(* CoDeSys 2.3.9.48 project: LevelControlTanks.pro *)
(* Libraries: Standard.lib 8.11.10 11:37:48, SYSLIBCALLBACK.LIB 8.11.10 11:37:48 *)

(* PLC configuration (modules and I/O channels)
K-Bus [K_Bus] node 0, in %IB0 out %QB0
Fieldbus variables [FB_VARS] node 1, in %IB0 out %QB0
Flag variables [FLAG_VARS] node 2, in %IB0 out %QB0
Modbus-Master [MB_MASTER] node 3, in %IB0 out %QB0
*)

(* Global variable list: Global_Variables *)
VAR_GLOBAL
			(*VALVES*)
	InletValve: BOOL;
	ConnectingValve: BOOL;
	OutletValve: BOOL;
			(*SENSORS 1=high, 2=ok, 3=low*)
	Tank1Sensors: ARRAY[1..NumSensors] OF BOOL;
	Tank2Sensors: ARRAY[1..NumSensors] OF BOOL;
			(*FAULT*)
	faultSensors1: BOOL;
	faultSensors2: BOOL;

			(*SENSOR STATEMENT*)
	sensorStatementINTTank1: INT;
	sensorStatementINTTank2: INT;
	sensorString1: STRING;
	sensorString2: STRING;
END_VAR

VAR_GLOBAL CONSTANT
	NumSensors: INT := 3;
	NumTanks: INT := 2;
END_VAR

(* POU PLC_PRG, ST *)
PROGRAM PLC_PRG
VAR
END_VAR
TANK1;
TANK2;
TanksFault;
TanksInletValve;
TanksOutletValves;
END_PROGRAM

(* POU TANK1, ST *)
PROGRAM TANK1
VAR
	i: INT := 1;
	k: INT := 0;
END_VAR
	(*TANK1*)
FOR i := 1 TO 2 DO
	sensorStatementINTTank1 := sensorsStatement(HighSensor:= Tank1Sensors[1], OKSensor:=Tank1Sensors[2], LowSensor := Tank1Sensors[3]);
END_FOR;

(*
		INT VALUES TANKS
	1: TANK IS NOT FILLED
	2: TANK IS LOW WATER LEVEL
	3: SENSORS FAULT (LOW)
	4: TANK IS ON OK WATER LEVEL
	5: SENSORS FAULT (LOW AND OKAY)
	6: SENSORS FAULT (OKAY)
	7: TANK IS FULL ENOUGH
*)

		(*TANK1*)
IF sensorStatementINTTank1 = 1 THEN
	sensorString1:= 'Tank1 is empty';
END_IF;

IF sensorStatementINTTank1 = 2 THEN
	sensorString1:= 'Tank 1 is on low water level';
END_IF;

IF sensorStatementINTTank1 = 3 THEN
	sensorString1:= 'Sensor fault tank 1(LowSensor)';
END_IF;

IF sensorStatementINTTank1 = 4 THEN
	sensorString1:= 'Tank1 is on OK water level';
END_IF;

IF sensorStatementINTTank1 = 5 THEN
	sensorString1:= 'Sensor fault tank 1(LowSensor, OKsensor)';
END_IF;

IF sensorStatementINTTank1 = 6 THEN
	sensorString1:= 'Sensor fault tank 1(OKSensor)';
END_IF;

IF sensorStatementINTTank1 = 7 THEN
	sensorString1:= 'Tank1 is full enough';
END_IF;
END_PROGRAM

(* POU sensorsStatement, ST *)
FUNCTION sensorsStatement : INT
VAR_INPUT
	Highsensor: BOOL;
	OkSensor: BOOL;
	LowSensor: BOOL;
END_VAR
VAR
END_VAR
(*
		INT VALUES TANKS
	1: TANK IS NOT FILLED
	2: TANK IS LOW WATER LEVEL
	3: SENSORS FAULT (LOW)
	4: TANK IS ON OK WATER LEVEL
	5: SENSORS FAULT (LOW AND OKAY)
	6: SENSORS FAULT (OKAY)
	7: TANK IS FULL ENOUGH
*)

IF HighSensor = FALSE AND OkSensor = FALSE AND LowSensor = FALSE THEN
	sensorsStatement := 1;
END_IF;
IF HighSensor = FALSE AND OkSensor = FALSE AND LowSensor = TRUE THEN sensorsStatement := 2;END_IF;
IF HighSensor = FALSE AND OkSensor = TRUE AND LowSensor = FALSE THEN sensorsStatement := 3; END_IF;
IF HighSensor = FALSE AND OkSensor = TRUE AND LowSensor = TRUE THEN sensorsStatement := 4;  END_IF;
IF HighSensor = TRUE AND OkSensor = FALSE AND LowSensor = FALSE THEN sensorsStatement := 5;END_IF;
IF HighSensor = TRUE AND OkSensor = FALSE AND LowSensor = TRUE THEN sensorsStatement := 6;END_IF;
IF HighSensor = TRUE AND OkSensor = TRUE AND LowSensor = FALSE THEN sensorsStatement := 3; END_IF;
IF HighSensor = TRUE AND OkSensor = TRUE  AND LowSensor = TRUE  THEN sensorsStatement := 7; END_IF;
END_FUNCTION

(* POU TANK2, ST *)
PROGRAM TANK2
VAR
	j: INT := 1;
END_VAR
	(*TANK2*)
FOR j := 1 TO 2 DO
	sensorStatementINTTank2 := sensorsStatement(HighSensor:= Tank2Sensors[1], OKSensor:=Tank2Sensors[2], LowSensor := Tank2Sensors[3]);
END_FOR;

(*
		INT VALUES TANKS
	1: TANK IS NOT FILLED
	2: TANK IS LOW WATER LEVEL
	3: SENSORS FAULT (LOW)
	4: TANK IS ON OK WATER LEVEL
	5: SENSORS FAULT (LOW AND OKAY)
	6: SENSORS FAULT (OKAY)
	7: TANK IS FULL ENOUGH
*)

		(*TANK2*)
IF sensorStatementINTTank2 = 1 THEN
	sensorString2:= 'Tank2 is empty';
END_IF;

IF sensorStatementINTTank2  = 2 THEN
	sensorString2:= 'Tank 2 is on low water level';
END_IF;

IF sensorStatementINTTank2  = 3 THEN
	sensorString2:= 'Sensor fault tank 2(LowSensor)';
END_IF;

IF sensorStatementINTTank2  = 4 THEN
	sensorString2:= 'Tank2 is on OK water level';
END_IF;

IF sensorStatementINTTank2  = 5 THEN
	sensorString2:= 'Sensor fault tank 2(LowSensor, OKsensor)';
END_IF;

IF sensorStatementINTTank2  = 6 THEN
	sensorString2:= 'Sensor fault tank 2(OKSensor)';
END_IF;

IF sensorStatementINTTank2  = 7 THEN
	sensorString2:= 'Tank2 is full enough';
END_IF;
END_PROGRAM

(* POU FunctionBlocks/TanksFault, CFC *)
PROGRAM TanksFault
VAR
END_VAR
VAR (* helpers for the ST form of the networks *)
	_t30 : BOOL;
	_t8 : BOOL;
	_t41 : BOOL;
	_t39 : BOOL;
END_VAR
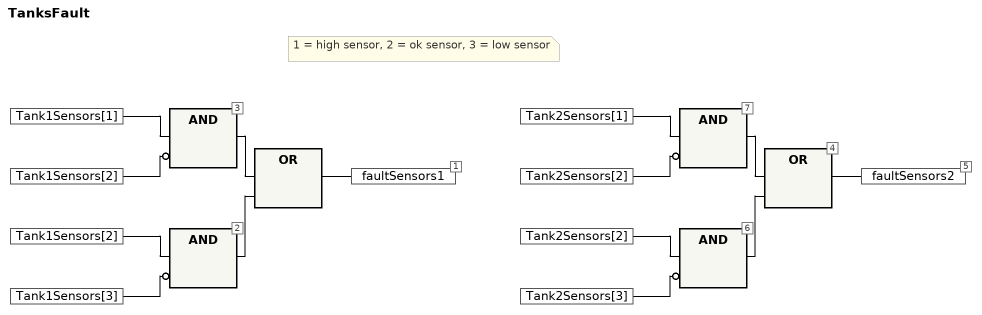
_CFC_ (* Continuous Function Chart, elements in execution order *)
(* 1 = high sensor, 2 = ok sensor, 3 = low sensor *)
#0 OR(#3, #2)
#1 faultSensors1 <= #0
#2 AND(Tank1Sensors[2], NOT Tank1Sensors[3])
#3 AND(Tank1Sensors[1], NOT Tank1Sensors[2])
#4 OR(#7, #6)
#5 faultSensors2 <= #4
#6 AND(Tank2Sensors[2], NOT Tank2Sensors[3])
#7 AND(Tank2Sensors[1], NOT Tank2Sensors[2])
_END_CFC_
(* the same logic as Structured Text *)
(* 1 = high sensor, 2 = ok sensor, 3 = low sensor *)
faultSensors1 := _t30 OR _t8;
_t8 := Tank1Sensors[2] AND NOT Tank1Sensors[3];
_t30 := Tank1Sensors[1] AND NOT Tank1Sensors[2];
faultSensors2 := _t41 OR _t39;
_t39 := Tank2Sensors[2] AND NOT Tank2Sensors[3];
_t41 := Tank2Sensors[1] AND NOT Tank2Sensors[2];
END_PROGRAM

(* POU FunctionBlocks/TanksInletValve, CFC *)
PROGRAM TanksInletValve
VAR
END_VAR
VAR (* helpers for the ST form of the networks *)
	_t30 : BOOL;
	_t8 : BOOL;
	_t52 : BOOL;
	_t50 : BOOL;
END_VAR
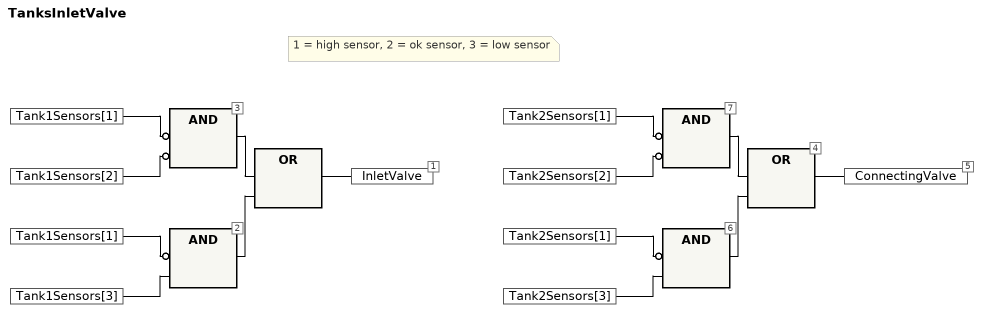
_CFC_ (* Continuous Function Chart, elements in execution order *)
(* 1 = high sensor, 2 = ok sensor, 3 = low sensor *)
#0 OR(#3, #2)
#1 InletValve <= #0
#2 AND(NOT Tank1Sensors[1], Tank1Sensors[3])
#3 AND(NOT Tank1Sensors[1], NOT Tank1Sensors[2])
#4 OR(#7, #6)
#5 ConnectingValve <= #4
#6 AND(NOT Tank2Sensors[1], Tank2Sensors[3])
#7 AND(NOT Tank2Sensors[1], NOT Tank2Sensors[2])
_END_CFC_
(* the same logic as Structured Text *)
(* 1 = high sensor, 2 = ok sensor, 3 = low sensor *)
InletValve := _t30 OR _t8;
_t8 := NOT Tank1Sensors[1] AND Tank1Sensors[3];
_t30 := NOT Tank1Sensors[1] AND NOT Tank1Sensors[2];
ConnectingValve := _t52 OR _t50;
_t50 := NOT Tank2Sensors[1] AND Tank2Sensors[3];
_t52 := NOT Tank2Sensors[1] AND NOT Tank2Sensors[2];
END_PROGRAM

(* POU FunctionBlocks/TanksOutletValves, CFC *)
PROGRAM TanksOutletValves
VAR
END_VAR
VAR (* helpers for the ST form of the networks *)
	_t30 : BOOL;
	_t8 : BOOL;
	_t61 : BOOL;
	_t59 : BOOL;
END_VAR
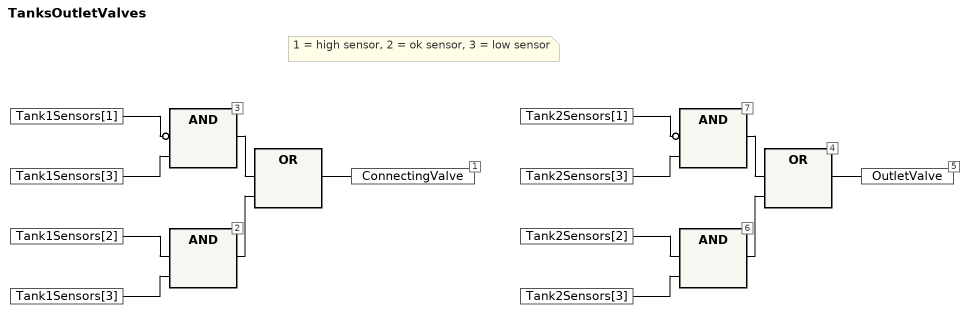
_CFC_ (* Continuous Function Chart, elements in execution order *)
(* 1 = high sensor, 2 = ok sensor, 3 = low sensor *)
#0 OR(#3, #2)
#1 ConnectingValve <= #0
#2 AND(Tank1Sensors[2], Tank1Sensors[3])
#3 AND(NOT Tank1Sensors[1], Tank1Sensors[3])
#4 OR(#7, #6)
#5 OutletValve <= #4
#6 AND(Tank2Sensors[2], Tank2Sensors[3])
#7 AND(NOT Tank2Sensors[1], Tank2Sensors[3])
_END_CFC_
(* the same logic as Structured Text *)
(* 1 = high sensor, 2 = ok sensor, 3 = low sensor *)
ConnectingValve := _t30 OR _t8;
_t8 := Tank1Sensors[2] AND Tank1Sensors[3];
_t30 := NOT Tank1Sensors[1] AND Tank1Sensors[3];
OutletValve := _t61 OR _t59;
_t59 := Tank2Sensors[2] AND Tank2Sensors[3];
_t61 := NOT Tank2Sensors[1] AND Tank2Sensors[3];
END_PROGRAM
